Fanuc KAREL source: ADD_DICT.kl

PROGRAM T
%NOLOCKGROUP
VAR
 v0 : STRING[40]
 v1 : STRING[40]
 v2 : STRING[40]
 v3 : INTEGER
 v4 : INTEGER
BEGIN
 ADD_DICT(v0, v1, v2, v3, v4)
END T
